// TIA Portal V16 export
// export: Created 2023-03-29T11:03:43.2021912Z, ExportSetting WithDefaults, DisplayName Totally Integrated Automation Portal, DisplayVersion V16 Update 6, DisplayName TIA Portal Version Control Interface, DisplayVersion V16 Update 2, DisplayName TIA Portal Openness, DisplayVersion V16 Update 6, DisplayName STEP 7 Professional, DisplayVersion V16 Update 6, DisplayName STEP 7 Safety, DisplayVersion V16, DisplayName WinCC Advanced, DisplayVersion V16 Update 6
DATA_BLOCK "Startegia_sterowania_DB"   // DB72
AUTHOR : rtecmer
VERSION : 0.1
// stored: AutoNumber true, DBAccessibleFromOPCUA true, InstanceOfName Startegia_sterowania, InstanceOfType FB
"Startegia_sterowania"
   // VAR
   //    tmp_time_1 : Bool;
   //    tmp_time_2 : Bool;
   //    tmp_time_3 : Bool;
   //    tmp_time_4 : Bool;
   // END_VAR
BEGIN
END_DATA_BLOCK
